FUNCTION "FC_Route_Supervisor" : Void
{ S7_Optimized_Access := 'TRUE' }
VERSION : 3.1
// ==============================================================================
// FC_Route_Supervisor - Супервізор маршрутів (Mailbox Pattern v3.1)
// ==============================================================================
// Версія: 3.2.2
// Дата: 2026-03-01
// ==============================================================================
// ЗМІНИ v3.2.2:
//   - Винесено магічні числа 12 та 64 у константи "ROUTES_COUNT" та "ROUTE_MAX_STEPS"
//
// ЗМІНИ v3.2.1:
//   [FIX-11] Cleanup: цикл FOR j обмежено MIN(RC_StepCount, 64).
//            RC_StepCount : USINT (0..255), RC_Steps : ARRAY[1..64].
//            FSM клампує stepCnt внутрішньо, але RC_StepCount у RouteExecutor
//            не змінює. Cleanup читав RC_StepCount напряму → j міг досягти 64+
//            → RC_Steps[j] виходив за межі масиву → потенційний OOB.
//
// ЗМІНИ v3.2.0:
//   [FIX-6] STOP_OP дозволено тільки з STARTING/RUNNING/STOPPING (не з VALIDATING).
//
//           ПРОБЛЕМА: VALIDATING входив до isActive → Supervisor копіював STOP_OP
//           у RouteExecutor → lastCmd ставав RT_CMD_STOP_OP ще до RUNNING.
//           Коли маршрут досягав RUNNING, stopOpEdge = FALSE (edge вже "спалений").
//           Повторні натискання STOP_OP також не давали ефекту — значення не змінювалось.
//           Зупинити маршрут можна було тільки через fault або GlobalSafetyStop.
//
//           РІШЕННЯ: окремий прапор isStoppable = STARTING OR RUNNING OR STOPPING.
//           У VALIDATING механізми ще не захоплені → STOP_OP там беззмістовний.
//           VALIDATING триває 1 скан-цикл → ігнорування STOP_OP непомітне для оператора.
//
// ЗМІНИ v3.1.0:
//   [FIX-5] Cleanup: не знуляє RC_StepCount поки механізми ще захоплені маршрутом.
//
//           ПРОБЛЕМА (v3.0): Cleanup знуляв RC_StepCount одразу після входу у ABORTED.
//           Це знищувало єдиний спосіб знайти механізми для retry CMD_RELEASE_OWNER:
//             - FSM ABORTED-retry: stepCnt = 0 → loop не запускався
//             - GlobalSafetyStop block: stepCnt = 0 → loop не запускався
//           Механізми залишались OWNER_ROUTE назавжди → deadlock (REJECT_BY_OWNER).
//
//           РІШЕННЯ: перед очищенням перевіряємо чи є ще OWNER_ROUTE в цього маршруту.
//           Якщо є — пропускаємо очищення; GlobalSafetyStop block або FSM ABORTED-retry
//           продовжують ретраювати CMD_RELEASE_OWNER кожен цикл (stepCnt збережено).
//           Коли всі механізми звільнені → Cleanup очищає → FSM → IDLE.
//
//           Сценарії що виправляє:
//             GlobalSafetyStop: механізм STS_STOPPING (секунди) → retry кожен цикл
//                               → STS_IDLE → ARB_OK → звільнено → Cleanup → IDLE ✓
//             STS_DISABLED під час STOPPING: Enable_OK відновлено → STS_IDLE
//                               → ARB_OK → звільнено → Cleanup → IDLE ✓
//
// ЗМІНИ v3.0.0:
//   [FIX-1] FC_RouteFSM читає GlobalSafetyStop, GlobalLocalManual напряму як глобальні теги ПЛК
//           (раніше параметри завжди передавались як FALSE)
//   [FIX-2] Невалідний RouteId → ACK + RETURN (раніше RETURN без ACK)
//           Mailbox більше не блокується назавжди
//   [FIX-3] REJECTED додано до Cleanup (раніше маршрут застрягав у REJECTED)
//           FSM може вийти з REJECTED → IDLE через RT_CMD_NONE
//   [FIX-4] STOP_OP для неактивного маршруту → RS_WARNING_IGNORED_CMD
//           (раніше "завжди дозволено" → сміття у RouteExecutor для REJECTED)
//
// v2.0.4:
//   FC_RouteFSM затирає RS_Warning кожного циклу для ВСІХ маршрутів
//   Рішення: Зберігати RS_Warning перед FSM і відновлювати після FSM
// ==============================================================================
   VAR_TEMP
      i : USInt;
      commitIn : UDInt;
      commitAck : UDInt;
      routeId : USInt;
      currentState : UInt;
      isActive : Bool;
      isStoppable : Bool;   // [FIX-6] STARTING OR RUNNING OR STOPPING (не VALIDATING)
      cmdAllowed : Bool;
      processedRouteId : USInt;
      pendingWarning : USInt;
      savedWarnings : Array[1.."ROUTES_COUNT"] of USInt;   // Зберегти RS_Warning
      j : Int;   // [FIX-5] ітератор кроків у Cleanup
      stepBound : Int;   // [FIX-11] верхня межа циклу (≤ROUTE_MAX_STEPS-1)
      innerSlot : UInt;   // [FIX-5] слот механізму у Cleanup
      routeAllReleased : Bool;   // [FIX-5] чи всі механізми звільнені
   END_VAR


BEGIN

	    // Ініціалізація
	    #processedRouteId := 0;
	    #pendingWarning := "RS_WARNING_OK";

	    // =========================================================
	    // 1. ЗБЕРЕГТИ RS_Warning перед FSM
	    // =========================================================
	    // ✅ КРИТИЧНО: FSM затирає RS_Warning кожного циклу
	    FOR #i := 1 TO "ROUTES_COUNT" DO
	        #savedWarnings[#i] := "DB_PlcToScada_RouteStatus".RoutesSts[#i].RS_Warning;
	    END_FOR;

	    // =========================================================
	    // 2. MAILBOX: Детект нової команди
	    // =========================================================
	    #commitIn := "DB_ScadaToPlc_RouteCmd".HDR_Commit;
	    #commitAck := "DB_PlcToScada_RouteStatus".ACK_CommitApplied;

	    IF #commitIn <> #commitAck THEN

	        // =========================================================
	        // 3. MAILBOX: Валідація RouteId
	        // =========================================================
	        #routeId := "DB_ScadaToPlc_RouteCmd".HDR_RouteId;

	        // Невалідний RouteId → ACK (mailbox не блокується) + RETURN
	        IF (#routeId < 1) OR (#routeId > "ROUTES_COUNT") THEN
	            "DB_PlcToScada_RouteStatus".ACK_CommitApplied := #commitIn;
	            "DB_PlcToScada_RouteStatus".ACK_RouteId := 0;
	            RETURN;
	        END_IF;

	        // =========================================================
	        // 4. MAILBOX: Перевірка стану маршруту
	        // =========================================================
	        #currentState := "DB_PlcToScada_RouteStatus".RoutesSts[#routeId].RS_State;

	        #isActive := (#currentState = "ROUTE_STS_VALIDATING") OR
	        (#currentState = "ROUTE_STS_STARTING") OR
	        (#currentState = "ROUTE_STS_RUNNING") OR
	        (#currentState = "ROUTE_STS_STOPPING");

	        // [FIX-6] STOP_OP дозволено тільки з STARTING/RUNNING/STOPPING
	        // У VALIDATING механізми ще не захоплені → STOP_OP беззмістовний
	        #isStoppable := (#currentState = "ROUTE_STS_STARTING") OR
	        (#currentState = "ROUTE_STS_RUNNING") OR
	        (#currentState = "ROUTE_STS_STOPPING");

	        #cmdAllowed := FALSE;

	        // Перевірка дозволеності команди
	        IF "DB_ScadaToPlc_RouteCmd".CMD_Route.RC_Cmd = "RT_CMD_START" THEN
	            IF #isActive THEN
	                // START для активного → ігнорувати з попередженням
	                #pendingWarning := "RS_WARNING_IGNORED_CMD";
	                #cmdAllowed := FALSE;
	            ELSE
	                // START для неактивного → дозволено
	                #pendingWarning := "RS_WARNING_OK";
	                #cmdAllowed := TRUE;
	            END_IF;

	        ELSIF "DB_ScadaToPlc_RouteCmd".CMD_Route.RC_Cmd = "RT_CMD_STOP_OP" THEN
	            IF #isStoppable THEN
	                // STOP_OP для STARTING/RUNNING/STOPPING — дозволено
	                #pendingWarning := "RS_WARNING_OK";
	                #cmdAllowed := TRUE;
	            ELSE
	                // STOP_OP для VALIDATING/IDLE/REJECTED/ABORTED — ігнорувати з попередженням
	                #pendingWarning := "RS_WARNING_IGNORED_CMD";
	                #cmdAllowed := FALSE;
	            END_IF;

	        ELSE
	            // RT_CMD_NONE або невідома команда
	            #cmdAllowed := FALSE;
	        END_IF;

	        // =========================================================
	        // 5. MAILBOX: Копіювання команди у RouteExecutor
	        // =========================================================
	        IF #cmdAllowed THEN
	            // [FIX-STOP] При STOP_OP НЕ затираємо RC_StepCount і RC_Steps!
	            // Вони містять активні кроки маршруту, які FSM використовує при STOPPING
	            IF "DB_ScadaToPlc_RouteCmd".CMD_Route.RC_Cmd = "RT_CMD_STOP_OP" THEN
	                // Тільки оновлюємо команду, шаги залишаються з START
	                "DB_Plc_RouteExecutor".Routes[#routeId].RC_Cmd := "RT_CMD_STOP_OP";
	            ELSE
	                // START або інші команди — повна копія
	                "DB_Plc_RouteExecutor".Routes[#routeId] := "DB_ScadaToPlc_RouteCmd".CMD_Route;
	            END_IF;
	        END_IF;

	        // =========================================================
	        // 6. MAILBOX: Підтвердження (ACK)
	        // =========================================================
	        "DB_PlcToScada_RouteStatus".ACK_CommitApplied := #commitIn;
	        "DB_PlcToScada_RouteStatus".ACK_RouteId := #routeId;

	        // Запам'ятати який маршрут обробили
	        #processedRouteId := #routeId;

	    END_IF;

	    // =========================================================
	    // 7. FSM: Виконання всіх маршрутів
	    // =========================================================
	    FOR #i := 1 TO "ROUTES_COUNT" DO

	        "FC_RouteFSM"(
	                      RouteIdx := INT_TO_USINT(#i),
	                      Cmd := "DB_Plc_RouteExecutor".Routes[#i],
	                      Mechs := "DB_Mechs".Mechs,
	                      Fsm := "DB_Plc_RouteFsm".RoutesFsm[#i],
	                      Sts => "DB_PlcToScada_RouteStatus".RoutesSts[#i]
	        );

	    END_FOR;

	    // =========================================================
	    // 8. ✅ ВІДНОВИТИ RS_Warning після FSM
	    // =========================================================
	    FOR #i := 1 TO "ROUTES_COUNT" DO
	        IF #i = #processedRouteId THEN
	            // Для обробленого маршруту → встановити новий Warning
	            "DB_PlcToScada_RouteStatus".RoutesSts[#i].RS_Warning := #pendingWarning;
	        ELSE
	            // Для інших маршрутів → відновити збережений Warning
	            "DB_PlcToScada_RouteStatus".RoutesSts[#i].RS_Warning := #savedWarnings[#i];
	        END_IF;
	    END_FOR;

	    // =========================================================
	    // 9. CLEANUP: Очищення RouteExecutor після завершення
	    // =========================================================
	    FOR #i := 1 TO "ROUTES_COUNT" DO
	        // Пропустити маршрут, який щойно отримав нову команду
	        IF #i = #processedRouteId THEN
	            CONTINUE;
	        END_IF;

	        #currentState := "DB_PlcToScada_RouteStatus".RoutesSts[#i].RS_State;

	        // Очищати маршрути у фінальних станах (REJECTED включено — без цього FSM застряє)
	        IF (#currentState = "ROUTE_STS_ABORTED") OR (#currentState = "ROUTE_STS_IDLE")
	            OR (#currentState = "ROUTE_STS_REJECTED") THEN

	            // [FIX-5] Перевірити чи є ще механізми що належать цьому маршруту.
	            //
	            // Якщо є — НЕ очищати RC_StepCount. Це зберігає список слотів живим для:
	            //   - GlobalSafetyStop block: ретраює CMD_RELEASE_OWNER кожен цикл
	            //     (поки GlobalSafetyStop активний і safetyHit = TRUE блокує FSM)
	            //   - FSM ABORTED retry: ретраює коли safetyHit = FALSE
	            //   Обидва варіанти завершаться успішно коли механізм досягне STS_IDLE/FAULT.
	            //
	            // Після того як всі механізми звільнені → Cleanup нулює → FSM → IDLE.
	            //
	            // Захист: innerSlot > MECHS_COUNT → пропускаємо (невалідний слот не читаємо).
	            #routeAllReleased := TRUE;
	            #stepBound := USINT_TO_INT("DB_Plc_RouteExecutor".Routes[#i].RC_StepCount);
	            IF #stepBound > "ROUTE_MAX_STEPS" THEN
	                #stepBound := "ROUTE_MAX_STEPS";
	            END_IF;
	            FOR #j := 1 TO #stepBound DO
	                #innerSlot := "DB_Plc_RouteExecutor".Routes[#i].RC_Steps[#j].RS_Slot;
	                IF #innerSlot <= "MECHS_COUNT" THEN
	                    IF ("DB_Mechs".Mechs[#innerSlot].OwnerCur = "OWNER_ROUTE") AND
	                        ("DB_Mechs".Mechs[#innerSlot].OwnerCurId = INT_TO_UINT(#i)) THEN
	                        #routeAllReleased := FALSE;
	                        EXIT;
	                    END_IF;
	                END_IF;
	            END_FOR;

	            IF #routeAllReleased THEN
	                "DB_Plc_RouteExecutor".Routes[#i].RC_Cmd := "RT_CMD_NONE";
	                "DB_Plc_RouteExecutor".Routes[#i].RC_StepCount := 0;
	            END_IF;

	        END_IF;
	    END_FOR;

END_FUNCTION

